// TIA Portal V20 export
TYPE "typeCmControlNodeBrakeTest"
// stored: Namespace Unit1.Em5
   STRUCT
      transferPnPLeftAxisZ : "LER_typeBrakeTestEmControlNodes";
      transferPnPRightAxisZ : "LER_typeBrakeTestEmControlNodes";
   END_STRUCT;
END_TYPE
